SUBAPPLICATION Button_IE_1 (* 1 Button-Objekt, liest ein konfigurierbares Event (ButtonActivationCode, z.B. BT_PRESSED_LATCHED) als reines IND-Event - duenner Wrapper um Button_IE, analog zu Aux_IE_1/Softkey_IE_1 (Konvention in diesem Projekt: die isobus-IE-Bausteine werden nie roh inline verwendet, immer gewrappt). *)
  (* Standard: 61499-2 *)
  (* Version 1.0, 2026-09-29, Franz Höpfinger, initial implementation, analog zu Aux_IE_1/Softkey_IE_1 *)
  PACKAGE MyLib::sys;
  IMPORT isobus::UT::Q::const::IDs::ID_NULL;
  IMPORT isobus::UT::io::Button::ButtonActivationCode::Invalid;
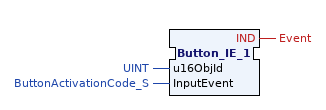
  EVENT_OUTPUT
    IND; (* Feuert wenn das konfigurierte InputEvent auftritt *)
  END_EVENT
  VAR_INPUT
    u16ObjId : UINT := ID_NULL; (* Object ID Button *)
    InputEvent : isobus::UT::io::Button::ButtonActivationCode_S := Invalid; (* z.B. BT_PRESSED_LATCHED, BT_RELEASED_UNLATCHED *)
  END_VAR
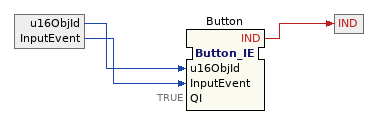
  FBS
    Button : isobus::UT::io::Button::Button_IE(QI := TRUE);
  END_FBS
  EVENT_CONNECTIONS
    Button.IND TO IND;
  END_CONNECTIONS
  DATA_CONNECTIONS
    u16ObjId TO Button.u16ObjId;
    InputEvent TO Button.InputEvent;
  END_CONNECTIONS
END_SUBAPPLICATION
